FUNCTION_BLOCK FB_SlitPairV2
VAR_INPUT
    ID_positiveAxis : UINT;
    ID_negativeAxis : UINT;
    ID_gapSizeAxis : UINT;
    ID_gapCentreAxis : UINT;
    
    Enable : BOOL;
    Reset : BOOL;
    EncoderScaling : LREAL := 10000;
END_VAR
VAR_OUTPUT    
END_VAR
VAR
    GapSizeEncoder AT %Q* : UDINT:=0;
    GapCentreEncoder AT %Q* : UDINT:=0;
    fGapSize : LREAL;
    fGapCentre : LREAL;
    
    setpointGenEnable_positiveAxis : MC_ExtSetPointGenEnable;    
    setpointGenEnable_negativeAxis : MC_ExtSetPointGenEnable;
    setpointGenEnable_gapSizeAxis : MC_ExtSetPointGenEnable;
    setpointGenEnable_gapCentreAxis : MC_ExtSetPointGenEnable;
    
    setpointGenDisable_positiveAxis : MC_ExtSetPointGenDisable;    
    setpointGenDisable_negativeAxis : MC_ExtSetPointGenDisable;
    setpointGenDisable_gapSizeAxis : MC_ExtSetPointGenDisable;
    setpointGenDisable_gapCentreAxis : MC_ExtSetPointGenDisable;
    
    posSetpoint_positiveAxis : LREAL;
    posSetpoint_negativeAxis : LREAL;
    posSetpoint_gapSizeAxis : LREAL;
    posSetpoint_gapCentreAxis : LREAL;
    
    veloSetpoint_positiveAxis : LREAL;
    veloSetpoint_negativeAxis : LREAL;
    veloSetpoint_gapSizeAxis : LREAL;
    veloSetpoint_gapCentreAxis : LREAL;
    
    dir_positiveAxis : DINT;
    dir_negativeAxis : DINT;
    dir_gapSizeAxis : DINT;
    dir_gapCentreAxis : DINT;
    
    iState : E_SlitPairStatesV2 := E_SlitPairStatesV2.INIT;
    
    internalReset : BOOL;
    
END_VAR

//Setup instructions
//Virtual encoder mask needs to be 0xFFFFFFFF

actVirtualAxisPositions();
GVL.astAxes[ID_gapSizeAxis].stConfig.eHomeSeq:= E_HomingRoutines.eHomeDirect;
GVL.astAxes[ID_gapCentreAxis].stConfig.eHomeSeq:= E_HomingRoutines.eHomeDirect;
GVL.astAxes[ID_gapSizeAxis].stConfig.fHomePosition:= fGapSize;
GVL.astAxes[ID_gapCentreAxis].stConfig.fHomePosition:= fGapCentre;

//What do we need

//Limit logic
actVirtualAxisLimits();
//Enable Logic
actVirtualAxisEnable();
//Call spGenerator FBs
actGeneratorEnableDisable();
//Calculate position setpoints
actCalculateSetpointPositions();
//Calculate velocity setpoints
actCalculateSetpointVelocities();
//Calculate directions
actCalculateSetpointDirections();

//We're only going to care about errors that stop motion!
IF GVL.astAxes[ID_positiveAxis].Axis.Status.ErrorStop OR GVL.astAxes[ID_negativeAxis].Axis.Status.ErrorStop OR GVL.astAxes[ID_gapSizeAxis].Axis.Status.ErrorStop OR GVL.astAxes[ID_gapCentreAxis].Axis.Status.ErrorStop THEN
    iState:= E_SlitPairStatesV2.ERROR_INIT;
END_IF

//Internal Reset linked to any axis reset
internalReset := Reset OR GVL.astAxes[ID_positiveAxis].stControl.bReset OR GVL.astAxes[ID_negativeAxis].stControl.bReset OR GVL.astAxes[ID_gapSizeAxis].stControl.bReset OR GVL.astAxes[ID_gapCentreAxis].stControl.bReset;

//State machine (with error handling and reset logic) - WHAT ABOUT HOMING?
IF Enable THEN
    CASE istate OF
        E_SlitPairStatesV2.INIT:
            IF GVL.astAxes[ID_positiveAxis].stStatus.bHomed AND GVL.astAxes[ID_negativeAxis].stStatus.bHomed THEN
                GVL.astAxes[ID_gapSizeAxis].stControl.eCommand:= E_MotionFunctions.eHome;
                GVL.astAxes[ID_gapSizeAxis].stControl.bExecute:= TRUE;
                GVL.astAxes[ID_gapcentreAxis].stControl.eCommand:= E_MotionFunctions.eHome;
                GVL.astAxes[ID_gapcentreAxis].stControl.bExecute:= TRUE;
                iState:=E_SlitPairStatesV2.WAIT_FOR_HOMED;
            ELSE
                iState:=E_SlitPairStatesV2.OPERATIONAL;
			END_IF
                     
        E_SlitPairStatesV2.WAIT_FOR_HOMED:
            IF GVL.astAxes[ID_gapSizeAxis].stStatus.bHomed AND GVL.astAxes[ID_gapCentreAxis].stStatus.bHomed THEN
                iState:=E_SlitPairStatesV2.OPERATIONAL;
			END_IF
       
        E_SlitPairStatesV2.OPERATIONAL:
            IF GVL.astAxes[ID_gapSizeAxis].stStatus.bMoving OR GVL.astAxes[ID_gapCentreAxis].stStatus.bMoving THEN
                iState:=E_SlitPairStatesV2.ENABLE_REAL_GENERATORS;
			END_IF
            IF GVL.astAxes[1].stStatus.bMoving OR GVL.astAxes[2].stStatus.bMoving THEN
                iState:=E_SlitPairStatesV2.ENABLE_VIRTUAL_GENERATORS;
            END_IF
            
        E_SlitPairStatesV2.ENABLE_REAL_GENERATORS:
            setpointGenEnable_positiveAxis.Execute:=TRUE;
            setpointGenEnable_negativeAxis.Execute:=TRUE;
            iState:=E_SlitPairStatesV2.WAIT_FOR_VIRTUAL_MOVE_DONE;
            
        E_SlitPairStatesV2.WAIT_FOR_VIRTUAL_MOVE_DONE:
            IF NOT(GVL.astAxes[ID_gapSizeAxis].stStatus.bMoving OR GVL.astAxes[ID_gapCentreAxis].stStatus.bMoving) THEN
                iState:=E_SlitPairStatesV2.DISABLE_REAL_GENERATORS;
			END_IF
            
        E_SlitPairStatesV2.DISABLE_REAL_GENERATORS:
            setpointGenDisable_positiveAxis.Execute:=TRUE;
            setpointGenDisable_negativeAxis.Execute:=TRUE;
            iState:=E_SlitPairStatesV2.OPERATIONAL;
            
        E_SlitPairStatesV2.ENABLE_VIRTUAL_GENERATORS:
            setpointGenEnable_gapSizeAxis.Execute :=TRUE;
            setpointGenEnable_gapCentreAxis.Execute:=TRUE;
            iState:=E_SlitPairStatesV2.WAIT_FOR_REAL_MOVE_DONE;
            
        E_SlitPairStatesV2.WAIT_FOR_REAL_MOVE_DONE:
            IF NOT(GVL.astAxes[1].stStatus.bMoving OR GVL.astAxes[2].stStatus.bMoving) THEN
                iState:=E_SlitPairStatesV2.DISABLE_VIRTUAL_GENERATORS;
			END_IF
            
        E_SlitPairStatesV2.DISABLE_VIRTUAL_GENERATORS:
            setpointGenDisable_gapSizeAxis.Execute :=TRUE;
            setpointGenDisable_gapCentreAxis.Execute:=TRUE;
            iState:=E_SlitPairStatesV2.OPERATIONAL;
            
        E_SlitPairStatesV2.ERROR_INIT:
            IF internalReset THEN
                GVL.astAxes[ID_positiveAxis].stControl.bReset := TRUE;
                GVL.astAxes[ID_negativeAxis].stControl.bReset := TRUE;
                GVL.astAxes[ID_gapSizeAxis].stControl.bReset := TRUE;
                GVL.astAxes[ID_gapCentreAxis].stControl.bReset := TRUE;
                iState:= E_SlitPairStatesV2.INIT;
			END_IF
    
	END_CASE
END_IF


//Feed externalsetpoint generators
MC_ExtSetPointGenFeed(Axis:= GVL.astAxes[ID_positiveAxis].Axis, Position:= posSetpoint_positiveAxis, Velocity:= veloSetpoint_positiveAxis, Acceleration:= 0, Direction:= dir_positiveAxis);
MC_ExtSetPointGenFeed(Axis:= GVL.astAxes[ID_negativeAxis].Axis, Position:= posSetpoint_negativeAxis, Velocity:= veloSetpoint_negativeAxis, Acceleration:= 0, Direction:= dir_negativeAxis);
MC_ExtSetPointGenFeed(Axis:= GVL.astAxes[ID_gapSizeAxis].Axis, Position:= posSetpoint_gapSizeAxis, Velocity:= veloSetpoint_gapSizeAxis, Acceleration:= 0, Direction:= dir_gapSizeAxis);
MC_ExtSetPointGenFeed(Axis:= GVL.astAxes[ID_gapCentreAxis].Axis, Position:= posSetpoint_gapCentreAxis, Velocity:= veloSetpoint_gapCentreAxis, Acceleration:= 0, Direction:= dir_gapCentreAxis);

ACTION actCalculateSetpointDirections:
IF veloSetpoint_positiveAxis >0 THEN
    dir_positiveAxis := 1; //moving forward
ELSIF veloSetpoint_positiveAxis <0 THEN
    dir_positiveAxis := -1; //moving backward
ELSE
    dir_positiveAxis := 0; //stationary
END_IF

IF veloSetpoint_negativeAxis >0 THEN
    dir_negativeAxis := 1; //moving forward
ELSIF veloSetpoint_negativeAxis <0 THEN
    dir_negativeAxis := -1; //moving backward
ELSE
    dir_negativeAxis := 0; //stationary
END_IF

IF veloSetpoint_gapSizeAxis >0 THEN
    dir_gapSizeAxis := 1; //moving forward
ELSIF veloSetpoint_gapSizeAxis <0 THEN
    dir_gapSizeAxis := -1; //moving backward
ELSE
    dir_gapSizeAxis := 0; //stationary
END_IF

IF veloSetpoint_gapCentreAxis >0 THEN
    dir_gapCentreAxis := 1; //moving forward
ELSIF veloSetpoint_gapCentreAxis <0 THEN
    dir_gapCentreAxis := -1; //moving backward
ELSE
    dir_gapCentreAxis := 0; //stationary
END_IF
END_ACTION

ACTION actCalculateSetpointPositions:
posSetpoint_positiveAxis := GVL.astAxes[ID_gapCentreAxis].Axis.NcToPlc.SetPos + (GVL.astAxes[ID_gapSizeAxis].Axis.NcToPlc.SetPos/2);
posSetpoint_negativeAxis := GVL.astAxes[ID_gapCentreAxis].Axis.NcToPlc.SetPos - (GVL.astAxes[ID_gapSizeAxis].Axis.NcToPlc.SetPos/2);
posSetpoint_gapSizeAxis := GVL.astAxes[ID_positiveAxis].Axis.NcToPlc.SetPos - GVL.astAxes[ID_negativeAxis].Axis.NcToPlc.SetPos;
posSetpoint_gapCentreAxis := (GVL.astAxes[ID_positiveAxis].Axis.NcToPlc.SetPos + GVL.astAxes[ID_negativeAxis].Axis.NcToPlc.SetPos) / 2;
END_ACTION

ACTION actCalculateSetpointVelocities:
veloSetpoint_positiveAxis := GVL.astAxes[ID_gapCentreAxis].Axis.NcToPlc.SetVelo +(GVL.astAxes[ID_gapSizeAxis].Axis.NcToPlc.SetVelo/2);
veloSetpoint_negativeAxis := GVL.astAxes[ID_gapCentreAxis].Axis.NcToPlc.SetVelo -(GVL.astAxes[ID_gapSizeAxis].Axis.NcToPlc.SetVelo/2);
veloSetpoint_gapSizeAxis := GVL.astAxes[ID_positiveAxis].Axis.NcToPlc.SetVelo - GVL.astAxes[ID_negativeAxis].Axis.NcToPlc.SetVelo;
veloSetpoint_gapCentreAxis := GVL.astAxes[ID_positiveAxis].Axis.NcToPlc.SetVelo + GVL.astAxes[ID_negativeAxis].Axis.NcToPlc.SetVelo;
END_ACTION

ACTION actGeneratorEnableDisable:
setpointGenEnable_positiveAxis(Axis:= GVL.astAxes[ID_positiveAxis].Axis);
setpointGenEnable_positiveAxis.Execute:= FALSE;

setpointGenEnable_negativeAxis(Axis:= GVL.astAxes[ID_negativeAxis].Axis);
setpointGenEnable_negativeAxis.Execute:= FALSE;

setpointGenEnable_gapSizeAxis(Axis:= GVL.astAxes[ID_gapSizeAxis].Axis);
setpointGenEnable_gapSizeAxis.Execute:= FALSE;

setpointGenEnable_gapCentreAxis(Axis:= GVL.astAxes[ID_gapCentreAxis].Axis);
setpointGenEnable_gapCentreAxis.Execute:= FALSE;


setpointGenDisable_positiveAxis(Axis:= GVL.astAxes[ID_positiveAxis].Axis);
setpointGenDisable_positiveAxis.Execute:= FALSE;

setpointGenDisable_negativeAxis(Axis:= GVL.astAxes[ID_negativeAxis].Axis);
setpointGenDisable_negativeAxis.Execute:= FALSE;

setpointGenDisable_gapSizeAxis(Axis:= GVL.astAxes[ID_gapSizeAxis].Axis);
setpointGenDisable_gapSizeAxis.Execute:= FALSE;

setpointGenDisable_gapCentreAxis(Axis:= GVL.astAxes[ID_gapCentreAxis].Axis);
setpointGenDisable_gapCentreAxis.Execute:= FALSE;
END_ACTION

ACTION actVirtualAxisEnable:
GVL.astAxes[ID_gapSizeAxis].stControl.bEnable := GVL.astAxes[ID_positiveAxis].stStatus.bEnabled AND GVL.astAxes[ID_negativeAxis].stStatus.bEnabled;
GVL.astAxes[ID_gapCentreAxis].stControl.bEnable := GVL.astAxes[ID_positiveAxis].stStatus.bEnabled AND GVL.astAxes[ID_negativeAxis].stStatus.bEnabled;
END_ACTION

ACTION actVirtualAxisLimits:
GVL.astAxes[ID_gapSizeAxis].stInputs.bLimitFwd:= GVL.astAxes[ID_positiveAxis].stStatus.bFwEnabled AND GVL.astAxes[ID_negativeAxis].stStatus.bBwEnabled;
GVL.astAxes[ID_gapSizeAxis].stInputs.bLimitBwd:= GVL.astAxes[ID_positiveAxis].stStatus.bBwEnabled AND GVL.astAxes[ID_negativeAxis].stStatus.bFwEnabled;

GVL.astAxes[ID_gapCentreAxis].stInputs.bLimitFwd:= GVL.astAxes[ID_positiveAxis].stStatus.bFwEnabled AND GVL.astAxes[ID_negativeAxis].stStatus.bFwEnabled;
GVL.astAxes[ID_gapCentreAxis].stInputs.bLimitBwd:= GVL.astAxes[ID_positiveAxis].stStatus.bBwEnabled AND GVL.astAxes[ID_negativeAxis].stStatus.bBwEnabled;
END_ACTION

ACTION actVirtualAxisPositions:
(*Calculate virtual axis positions and convert to UDINT.
Conversion to UDINT is prohibited if it would exceed UDINT max value of 4,294,967,295.
If this is not done, it can cause overflow when connected to the encoder input and hard-crash the PLC which will only recover with a power cycle.
To preserve decimal position data of the LREAL (i.e. anything <1mm) it is necessary to scale the value before converting to UDINT.
This can be reversed with the correct scaling at the NC encoder level.
*)
fGapSize := GVL.astAxes[ID_positiveAxis].stStatus.fActPosition - GVL.astAxes[ID_negativeAxis].stStatus.fActPosition;
fGapCentre := (GVL.astAxes[ID_positiveAxis].stStatus.fActPosition + GVL.astAxes[ID_negativeAxis].stStatus.fActPosition) / 2;


    IF ABS(fGapSize) < 100000 THEN
        GapSizeEncoder := LREAL_TO_UDINT(fGapSize*EncoderScaling);
    END_IF
    IF ABS(fGapCentre) < 100000 THEN
        GapCentreEncoder := LREAL_TO_UDINT(fGapCentre*EncoderScaling);
    END_IF
END_ACTION

END_FUNCTION_BLOCK

(* stored: Version 1.1.0.1, ProductVersion 3.1.4024.5
   POU FB_SlitPairV2: Id {ff4013b1-472a-4f42-a6c8-2711712ac06d}, SpecialFunc None
   Action actCalculateSetpointDirections: Id {7783e346-7fab-40d5-bab7-fe46a8c2f785}
   Action actCalculateSetpointPositions: Id {08e35b97-914a-4ccc-a3af-6b7cd8e60439}
   Action actCalculateSetpointVelocities: Id {59813eea-6905-4661-a8f3-10b16a472979}
   Action actGeneratorEnableDisable: Id {d59f6d39-50eb-4cb0-8d9d-b62df150c5a5}
   Action actVirtualAxisEnable: Id {d8729d12-361d-472b-8974-5b566dad7d06}
   Action actVirtualAxisLimits: Id {436d835a-8846-47e9-922d-a1df63469a25}
   Action actVirtualAxisPositions: Id {4ef557a2-3171-4a03-98ba-14f2cd3ef5ec} *)
